PROGRAM SevenDayOnOffConf
VAR

	bOver2ndLimitAlarmOccur: BOOL;


END_VAR

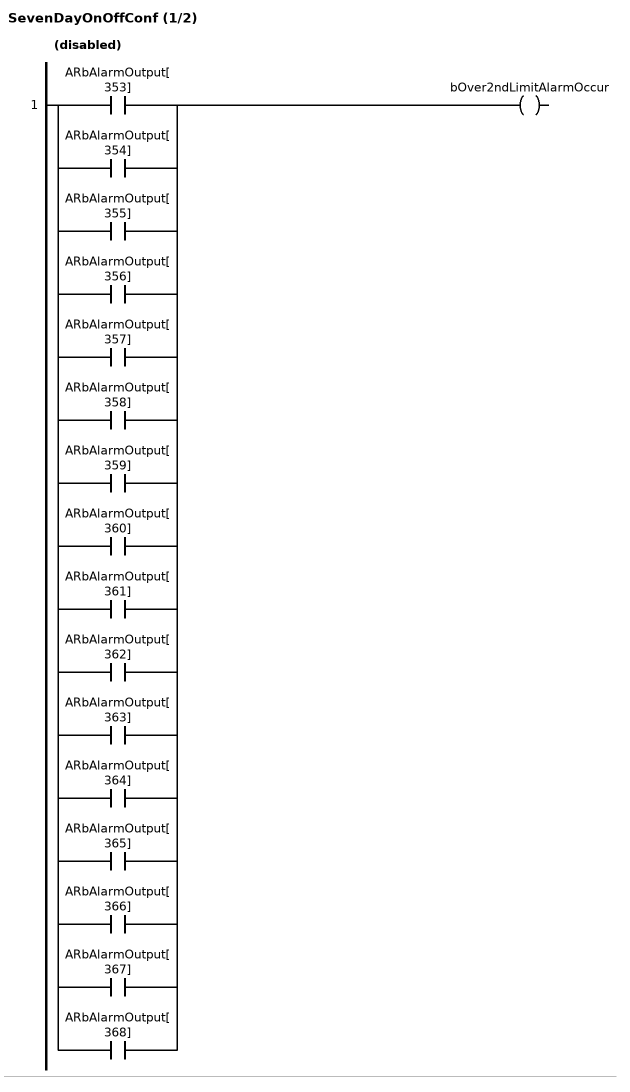
// NETWORK 1 (disabled)
// bOver2ndLimitAlarmOccur := ARbAlarmOutput[353] OR ARbAlarmOutput[354] OR ARbAlarmOutput[355] OR ARbAlarmOutput[356] OR ARbAlarmOutput[357] OR ARbAlarmOutput[358] OR ARbAlarmOutput[359] OR ARbAlarmOutput[360] OR ARbAlarmOutput[361] OR ARbAlarmOutput[362] OR ARbAlarmOutput[363] OR ARbAlarmOutput[364] OR ARbAlarmOutput[365] OR ARbAlarmOutput[366] OR ARbAlarmOutput[367] OR ARbAlarmOutput[368];

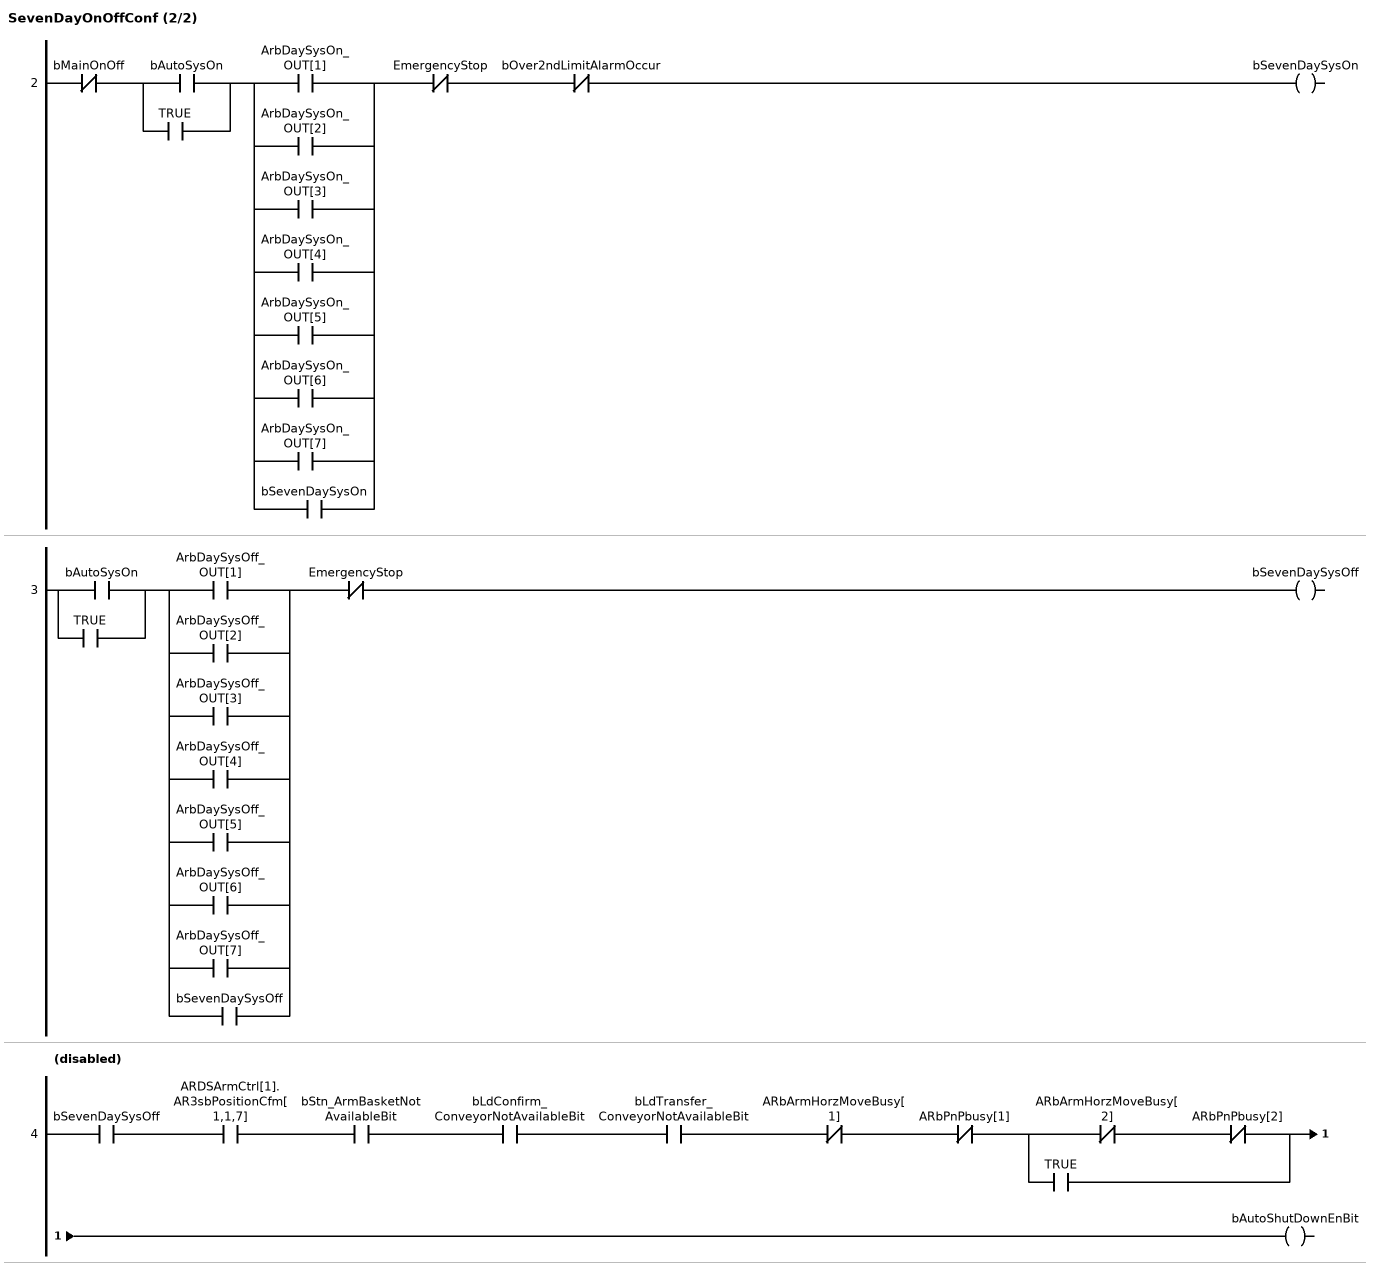
// NETWORK 2
bSevenDaySysOn := (NOT bMainOnOff AND (bAutoSysOn OR TRUE) AND (ArbDaySysOn_OUT[1] OR ArbDaySysOn_OUT[2] OR ArbDaySysOn_OUT[3] OR ArbDaySysOn_OUT[4] OR ArbDaySysOn_OUT[5] OR ArbDaySysOn_OUT[6] OR ArbDaySysOn_OUT[7] OR bSevenDaySysOn)) AND NOT EmergencyStop AND NOT bOver2ndLimitAlarmOccur;

// NETWORK 3
bSevenDaySysOff := ((bAutoSysOn OR TRUE) AND (ArbDaySysOff_OUT[1] OR ArbDaySysOff_OUT[2] OR ArbDaySysOff_OUT[3] OR ArbDaySysOff_OUT[4] OR ArbDaySysOff_OUT[5] OR ArbDaySysOff_OUT[6] OR ArbDaySysOff_OUT[7] OR bSevenDaySysOff)) AND NOT EmergencyStop;

// NETWORK 4 (disabled)
// bAutoShutDownEnBit := bSevenDaySysOff AND ARDSArmCtrl[1].AR3sbPositionCfm[1,1,7] AND bStn_ArmBasketNotAvailableBit AND bLdConfirm_ConveyorNotAvailableBit AND bLdTransfer_ConveyorNotAvailableBit AND NOT ARbArmHorzMoveBusy[1] AND NOT ARbPnPbusy[1] AND (NOT ARbArmHorzMoveBusy[2] AND NOT ARbPnPbusy[2] OR TRUE);

END_PROGRAM

(* stored: Version 1.1.0.1, ProductVersion 3.1.4024.12
   POU SevenDayOnOffConf: Id {423bb112-67ea-4fa7-84e1-285f66cf5c42}, SpecialFunc None *)
